PROGRAM PRG_Questar
VAR
    fb_Ques_01 : FB_MotionStage;
    fb_Ques_02: FB_MotionStage;
    bInit : BOOl := TRUE;
END_VAR


IF ( bInit) THEN
    bInit := FALSE;
    Main.M17.bHardwareEnable := TRUE;
    Main.M17.bPowerSelf := TRUE;
    Main.M17.nBrakeMode := ENUM_StageBrakeMode.NO_BRAKE;
    Main.M17.nEnableMode := ENUM_StageEnableMode.DURING_MOTION;
    Main.M17.fVelocity := 0.1;

    Main.M18.bHardwareEnable := TRUE;
    Main.M18.bPowerSelf := TRUE;
    Main.M18.nBrakeMode := ENUM_StageBrakeMode.NO_BRAKE;
    Main.M18.nEnableMode := ENUM_StageEnableMode.DURING_MOTION;
    Main.M18.fVelocity := 0.1;


END_IF
//EPS??


fb_Ques_01(stMotionStage:=Main.M17);
fb_Ques_02(stMotionStage:=Main.M18);

END_PROGRAM

(* stored: Version 1.1.0.1
   POU PRG_Questar: Id {a13b4cbe-0334-43ca-a474-80a981d3c693}, SpecialFunc None *)
